// TIA Portal V19 export
DATA_BLOCK "M0940_PIDInterfaceDB"   // DB8
{ S7_Optimized_Access := 'TRUE' }
// stored: AutoNumber false, MemoryReserve 0
   VAR RETAIN
      PC : "M0940_PIDInterface";
      LC : "M0940_PIDInterface";
   END_VAR
BEGIN
   PC.PV := 0.0;
   PC.SP := 1.0;
   PC.EngUnitsMin := 0.0;
   PC.EngUnitsMax := 16.0;
   PC.P := -0.5;
   PC.I := T#15S;
   LC.PV := 0.0;
   LC.SP := 50.0;
   LC.EngUnitsMin := 0.0;
   LC.EngUnitsMax := 100.0;
   LC.P := 1.5;
   LC.I := T#25S;
END_DATA_BLOCK
